PROGRAM MAIN
VAR
	// More about context and tasks here: https://docs.tcopengroup.org/articles/TcOpenFramework/application.html
	_context : ModBusContext;
END_VAR

// This runs the context.
_context.Run();

END_PROGRAM

(* stored: Version 1.1.0.1, ProductVersion 3.1.4024.9
   POU MAIN: Id {4cb653d2-485a-437a-9c01-820cb0a55b64}, SpecialFunc None *)
